# B&R Automation Studio project smart_home
Automation Studio 4.9

## Configuration Config1

CPU X20CP0410, AutomationRuntime 6.5.1, Build 11.3.0, Vc 6.0.0

### Task classes (Cpu.sw)
```
Cyclic#4 (cycle 100000 us, tolerance 100000 us):
  Program <- Program.prg
Libraries: ArCan, runtime, brsystem, standard, AsBrStr, AsBrWStr
```

### Hardware
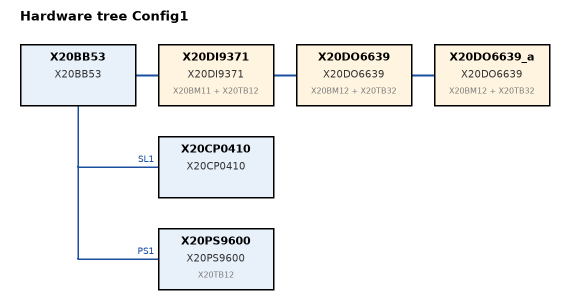
```
X20BB53 : X20BB53 v1.0.1.0
X20BM11 : X20BM11 v1.1.0.0  [X2X1 -> X20BB53.IF6]
X20BM12 : X20BM12 v1.1.0.0  [X2X1 -> X20BM11.X2X2]
X20BM12_a : X20BM12 v1.1.0.0  [X2X1 -> X20BM12.X2X2]
X20CP0410 : X20CP0410 v1.7.3.0  [SL -> X20BB53.SL1]
  Connector IF2:
    ActivateDevice = 1
  ConfigurationID = smart_home_Config1
  Simulation = 1
  TimerDeviceType = SWIOTIMER
  Cyclic1Duration = 10000
  Cyclic1Tolerance = 10000
  Cyclic2Duration = 20000
  Cyclic2Tolerance = 20000
  Cyclic3Duration = 50000
  Cyclic3Tolerance = 50000
  Cyclic4Duration = 100000
  Cyclic4Tolerance = 100000
  Cyclic5Duration = 200000
  Cyclic5Tolerance = 200000
  Cyclic6Duration = 500000
  Cyclic6Tolerance = 500000
  Cyclic7Duration = 1000000
  Cyclic7Tolerance = 1000000
  Cyclic8Duration = 10000
  Cyclic8Tolerance = 30000000
  FileDevice1
  FileDeviceName1 = USER
  FileDevicePath1 = USER_PATH
X20DI9371 : X20DI9371 v1.6.1.0  [SS1 -> X20TB12.SS; SL -> X20BM11.SL1]
X20DO6639 : X20DO6639 v1.2.2.0  [SS1 -> X20TB32.SS; SL -> X20BM12.SL1]
X20DO6639_a : X20DO6639 v1.2.2.0  [SS1 -> X20TB32_a.SS; SL -> X20BM12_a.SL1]
X20PS9600 : X20PS9600 v1.6.2.0  [PS -> X20BB53.PS1; SS1 -> X20TB12_a.SS]
X20TB12 : X20TB12 v1.0.0.0
X20TB12_a : X20TB12 v1.0.0.0
X20TB32 : X20TB32 v1.0.0.1
X20TB32_a : X20TB32 v1.0.0.1
```

## Logical view

Binary libraries used (declarations not repeated): operator, runtime, AsIecCon, ArCan, brsystem, standard, AsBrStr, AsBrWStr

### Global.typ
```iecst
TYPE
	hall : 	STRUCT
		light_h_1 : BOOL;
		light_h_2 : BOOL;
		light_h_3 : BOOL;
		door_h_main : BOOL;
		door_H_be : REFERENCE TO BOOL;
		door_H_liv : REFERENCE TO BOOL;
		door_H_bat : REFERENCE TO BOOL;
		door_H_ki : REFERENCE TO BOOL;
		swich_h_1 : BOOL;
		swich_h_2 : BOOL;
		swich_h_3 : BOOL;
		swich_h_4 : BOOL;
		swich_h_5 : BOOL;
		AC : BOOL;
	END_STRUCT;

		bed : 	STRUCT
		door_h_Be : REFERENCE TO BOOL;
		light_be_1 : BOOL;
		swich_be_1 : BOOL;
	END_STRUCT;

		liv :	STRUCT
		door_h_Liv : REFERENCE TO BOOL;
		light_liv_1 : BOOL;
		swich_liv_1 : BOOL;
		END_STRUCT;

		kit :	STRUCT
		door_h_Ki : REFERENCE TO BOOL;
		light_ki_1 : BOOL;
		light_ki_2 : BOOL;
		swich_ki_1 : BOOL;
		swich_ki_2 : BOOL;
		END_STRUCT;

		bat : STRUCT
		door_h_Bat : REFERENCE TO BOOL;
		light_bat_1 : BOOL;
		light_bat_2 : BOOL;
		swich_bat_1 : BOOL;
		flo_sen : BOOL;
		END_STRUCT;
END_TYPE
```

### Global.var
```iecst
VAR
	door_h_be : BOOL;
    door_h_liv : BOOL;
    door_h_bat : BOOL;
    door_h_ki : BOOL;
    hallway : hall;
    previous_halway : hall;
    bedroom : bed;
    previous_bedroom : bed;
    livingroom : liv;
    previous_livingroom : liv;
    kithen : kit;
    previous_kithem : kit;
    bathroom : bat;
    previous_bathroom : bat;
    status : UDINT;
    changes : BOOL;
    state_activ : BOOL;
    state_un_activ : BOOL;
END_VAR

VAR CONSTANT

END_VAR
```

### compile_flags.txt
```
# This file is auto-generated by ASX. Do not edit manually, as changes may be overwritten.
# If you need to manually edit this file and prevent automatic updates, add "# MANUAL EDIT" to the first line.
-I
C:\Program Files (x86)\BRAutomation\AS6\AS\gnuinst\V11.3.0\6.0\i686-elf\include\c++\11.3.0
-I
C:\Program Files (x86)\BRAutomation\AS6\AS\gnuinst\V11.3.0\6.0\i686-elf\include\c++\11.3.0\i686-elf
-I
C:\Program Files (x86)\BRAutomation\AS6\AS\gnuinst\V11.3.0\6.0\i686-elf\include\c++\11.3.0\backward
-I
C:\Program Files (x86)\BRAutomation\AS6\AS\gnuinst\V11.3.0\6.0\lib\gcc\i686-elf\11.3.0\include
-I
C:\Program Files (x86)\BRAutomation\AS6\AS\gnuinst\V11.3.0\6.0\lib\gcc\i686-elf\11.3.0\include-fixed
-I
C:\Program Files (x86)\BRAutomation\AS6\AS\gnuinst\V11.3.0\6.0\i686-elf\include
-I
c:\Praktyki\Smart_home\smart_home\Temp\Includes
-trigraphs
-fno-asm
-D
_DEFAULT_INCLUDES
-D
_SG4
--target=i686-elf
-fPIC
-Wall
```

### Program Logical/Program

#### Variables.var
```iecst
VAR
	i : INT;
	siezeof : FUB_TYPE;
END_VAR
```

#### Cyclic.st
```iecst
PROGRAM _CYCLIC

 IF brsmemcpy(ADR(hallway), ADR(previous_halway), SIZEOF(hallway)) >0 OR
    brsmemcpy(ADR(bedroom), ADR(previous_bedroom), SIZEOF(bedroom)) >0 OR
	brsmemcpy(ADR(livingroom), ADR(previous_livingroom), SIZEOF(livingroom)) >0 OR
	brsmemcpy(ADR(kithen), ADR(previous_kithem), SIZEOF(kithen)) >0 OR
	brsmemcpy(ADR(bathroom), ADR(previous_bathroom), SIZEOF(bathroom)) >0 THEN
		changes := TRUE
 END_IF;

	FOR i := 0 TO SIZEOF(hallway)/siezeof(hallway.AC) DO
		IF  arrHall[i] <> arrLastHall[i] THEN
			change := TRUE;
		END_IF;
	END_FOR
	IarrHallway
IF bedroom.swich_be_1 THEN
bedroom.light_be_1 := TRUE;
ELSE
bedroom.light_be_1 := FALSE;
END_IF;

IF livingroom.swich_liv_1 THEN
livingroom.light_liv_1 := TRUE;
ELSE
livingroom.light_liv_1 := FALSE;
END_IF;

IF bathroom.swich_bat_1 THEN
	bathroom.light_bat_1 := TRUE;
	bathroom.light_bat_2 := TRUE;
	ELSE
	bathroom.light_bat_1 := FALSE;
	bathroom.light_bat_2 := FALSE;
END_IF;

kithen.light_ki_1
AND
kithen.light_ki_2 := kithen.swich_ki_1
XOR
kithen.swich_ki_2;

hallway.light_h_1
AND
hallway.light_h_2
AND
hallway.light_h_3 := hallway.swich_h_1
XOR
hallway.swich_h_2
XOR
hallway.swich_h_3
XOR
hallway.swich_h_4
XOR
hallway.swich_h_5;

IF state_un_activ THEN
state_activ := FALSE;
hallway.light_h_1 := FALSE;
hallway.light_h_2 := FALSE;
hallway.light_h_3 := FALSE;
bedroom.light_be_1 := FALSE;
livingroom.light_liv_1 := FALSE;
kithen.light_ki_1 := FALSE;
kithen.light_ki_2 := FALSE;
bathroom.light_bat_1 := FALSE;
bathroom.light_bat_2 := FALSE;
END_IF;
IF changes THEN
state_activ := TRUE
END_IF;

END_PROGRAM
```

#### Init.st
```iecst
PROGRAM _INIT
	hallway.door_H_be := ADR(door_h_be);
	bedroom.door_h_Be := ADR(door_h_be);
	hallway.door_H_liv := ADR(door_h_liv);
	livingroom.door_h_Liv := ADR(door_h_liv);
	hallway.door_H_ki := ADR(door_h_ki);
	kithen.door_h_Ki := ADR(door_h_ki);
	hallway.door_H_bat := ADR(door_h_bat);
	bathroom.door_h_Bat := ADR(door_h_bat);
END_PROGRAM
```
